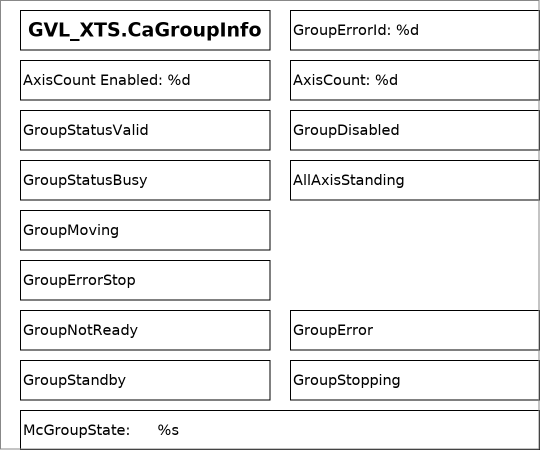
VISUALIZATION GROUP_VISU  // 540x450
    Rectangle (20,110 250x40), "GroupStatusValid", colour toggle: GVL_XTS.XtsTransportState[MAIN.nXpuSelected].GroupInfo.GroupStatusValid
    Rectangle (20,160 250x40), "GroupStatusBusy", colour toggle: GVL_XTS.XtsTransportState[MAIN.nXpuSelected].GroupInfo.GroupStatusBusy
    Rectangle (20,210 250x40), "GroupMoving", colour toggle: GVL_XTS.XtsTransportState[MAIN.nXpuSelected].GroupInfo.GroupMoving
    Rectangle (20,260 250x40), "GroupErrorStop", colour toggle: GVL_XTS.XtsTransportState[MAIN.nXpuSelected].GroupInfo.GroupErrorStop
    Rectangle (20,310 250x40), "GroupNotReady", colour toggle: GVL_XTS.XtsTransportState[MAIN.nXpuSelected].GroupInfo.GroupNotReady
    Rectangle (20,360 250x40), "GroupStandby", colour toggle: GVL_XTS.XtsTransportState[MAIN.nXpuSelected].GroupInfo.GroupStandby
    Rectangle (290,360 250x40), "GroupStopping", colour toggle: GVL_XTS.XtsTransportState[MAIN.nXpuSelected].GroupInfo.GroupStopping
    Rectangle (290,110 250x40), "GroupDisabled", colour toggle: GVL_XTS.XtsTransportState[MAIN.nXpuSelected].GroupInfo.GroupDisabled
    Rectangle (290,160 250x40), "AllAxisStanding", colour toggle: GVL_XTS.XtsTransportState[MAIN.nXpuSelected].GroupInfo.AllAxesStanding
    Rectangle (290,310 250x40), "GroupError", colour toggle: GVL_XTS.XtsTransportState[MAIN.nXpuSelected].GroupInfo.GroupError
    Rectangle (290,10 250x40), "GroupErrorId: %d", text variable: GVL_XTS.XtsTransportState[MAIN.nXpuSelected].GroupInfo.GroupErrorId
    Rectangle (290,60 250x40), "AxisCount: %d", text variable: GVL_XTS.XtsTransportState[MAIN.nXpuSelected].GroupInfo.AxisCount
    Rectangle (20,410 520x40), "McGroupState: %s", text variable: MAIN.sCaGroupState
    Rectangle (20,10 250x40), "GVL_XTS.CaGroupInfo"
    Rectangle (20,60 250x40), "AxisCount Enabled: %d", text variable: GVL_XTS.CaGroupInfo[MAIN.nXpuSelected].AxisCountEnabled
END_VISUALIZATION

(* stored: Version 1.1.0.1, ProductVersion 3.1.4026.12
   Visu GROUP_VISU: Id {9dcaf819-5ca7-43b4-8101-6ccb4d5cb710} *)
